INTERFACE I_RunnableTestFunctionBlock

METHOD RunTests : E_TestFunctionBlockRunState
END_METHOD

END_INTERFACE

(* stored: Version 1.1.0.1, ProductVersion 3.1.4022.12
   Itf I_RunnableTestFunctionBlock: Id {b4cb3522-b646-42db-9aab-52e064bbc290}
   Method RunTests: Id {984eeed7-7a78-402f-ae44-0c7d72008dda} *)
